(* IEC 61131-3 sources: volt/packages/volt-lsp-iec/test-corpus/bakon-nano/Device/Plc Logic/Application/POUs/FunctionBlocksAGM, 5 files *)

(* ---- ReadParametersFromAGM.pou ---- *)
FUNCTION_BLOCK ReadParametersFromAGM
VAR
	byStepper: BYTE;
	R_TRIG1: R_TRIG;
	bStartRead: BOOL;
	R_TRIG2: R_TRIG;
	LenzeParRead_LDC1: CIA405.SDO_READ4; (*TODO aanroep fixen CAA_Cia_405 en dan SDO_READ4*)
	Device : CIA405.DEVICE := 21;
	BLINK1: BLINK;
	TON1 :TON;
	byMasterNumber:BYTE:= 1;
	ptrByteArray : POINTER TO ARRAY[0..3] OF BYTE;
END_VAR
VAR_INPUT
	I_bEnable:BOOL;
END_VAR
VAR_OUTPUT
	bReady: BOOL;
END_VAR
VAR_IN_OUT
	Q_dwAGM_Status			: DWORD;
	Q_dwAGM_PowerLoss	: DWORD;
	Q_dwAGM_Frequency	: REAL;
	Q_dwAGM_ID				: DWORD;
END_VAR

%LANGUAGE ST
(*Create toggle for reading the parameters*)
BLINK1		(ENABLE:=I_bEnable ,
				 TIMELOW:=t#6s ,
				TIMEHIGH:=t#100ms,
				OUT=> );
R_TRIG1(CLK:=BLINK1.OUT);

IF R_TRIG1.Q THEN
	bStartRead:=TRUE;
END_IF

R_TRIG2(CLK:=LenzeParRead_LDC1.ERROR <> CIA405.CANOPEN_KERNEL_ERROR.CANOPEN_KERNEL_NO_ERROR);// OR LenzeParRead_LDC1.xTimeOut);(*TODO*)

IF NOT bStartRead OR R_TRIG2.Q OR NOT I_bEnable THEN
	byStepper:=0;
	bReady:=FALSE;
	bStartRead:=FALSE;
	LenzeParRead_LDC1(ENABLE:=FALSE);
	Q_dwAGM_ID := 0;
ELSE
	(*Alleen tijdens opstarten uitlezen*)
	CASE byStepper OF
	0:	(*Reset write FB*)
		bReady:=FALSE;
		TON1(IN:= FALSE);
		byStepper:=1;

	(*index 2003, generator status*)
	1:	LenzeParRead_LDC1(
		ENABLE:= FALSE,
		NETWORK :=byMasterNumber,
		Device:= Device,		 (* Adresse des Reglers *)
		Index:=8195,					(* Code *)
		SUBIndex:=0);				(* SubCode *)
		byStepper:=2;

	2:	LenzeParRead_LDC1(ENABLE:=TRUE,
								NETWORK:=ByMasterNumber);
		IF LenzeParRead_LDC1.CONFIRM THEN
			ptrByteArray := ADR(Q_dwAGM_Status);
			ptrByteArray^[0] := LenzeParRead_LDC1.DATA[1];
			ptrByteArray^[1] := LenzeParRead_LDC1.DATA[2];
			ptrByteArray^[2] := LenzeParRead_LDC1.DATA[3];
			ptrByteArray^[3] := LenzeParRead_LDC1.DATA[4];
			//Q_dwAGM_Status := SHL(SHL(SHL(LenzeParRead_LDC1.DATA[4],8) OR LenzeParRead_LDC1.DATA[3],8) OR LenzeParRead_LDC1.DATA[2],8) OR LenzeParRead_LDC1.DATA[1];	(* Codestelle wird gelesen *)
			LenzeParRead_LDC1(ENABLE:=FALSE);
			byStepper:=6;
		END_IF

	(*index 2008, Power loss*)
	6:	LenzeParRead_LDC1(
		ENABLE:= FALSE,
		Device:= Device,			(* Adresse des Reglers *)
		Index:=8200,						(* Code *)
		SubIndex:=0);					(* SubCode *)
		TON1(IN:=TRUE, PT:= t#1000ms);
		IF TON1.Q THEN
			byStepper:=8;
			TON1(IN:= FALSE);
		END_IF

	8:	LenzeParRead_LDC1(ENABLE:=TRUE,
								NETWORK:=1 );
		IF LenzeParRead_LDC1.CONFIRM THEN
			ptrByteArray := ADR(Q_dwAGM_PowerLoss);
			ptrByteArray^[0] := LenzeParRead_LDC1.DATA[1];
			ptrByteArray^[1] := LenzeParRead_LDC1.DATA[2];
			ptrByteArray^[2] := LenzeParRead_LDC1.DATA[3];
			ptrByteArray^[3] := LenzeParRead_LDC1.DATA[4];
			//Q_dwAGM_PowerLoss :=SHL(SHL(SHL(LenzeParRead_LDC1.DATA[4],8) OR LenzeParRead_LDC1.DATA[3],8) OR LenzeParRead_LDC1.DATA[2],8) OR LenzeParRead_LDC1.DATA[1];	(* Codestelle wird gelesen *)
			LenzeParRead_LDC1(ENABLE:=FALSE);
			byStepper:=12;
		END_IF

	(*index 2009, weld frequency*)
	12:	LenzeParRead_LDC1(
		Enable:= FALSE,
		NETWORK:=1,
		DEVICE:= Device,		(* Adresse des Reglers *)
		INDEX:=8201,					(* Code *)
		SUBINDEX:=0);				(* SubCode *)
		TON1(IN:=TRUE, PT:= t#1000ms);
		IF TON1.Q THEN
			byStepper:=14;
			TON1(IN:= FALSE);
		END_IF

	14:LenzeParRead_LDC1(ENABLE:=TRUE,
								NETWORK:=1);
		IF LenzeParRead_LDC1.CONFIRM THEN
			ptrByteArray := ADR(Q_dwAGM_Frequency);
			ptrByteArray^[0] := LenzeParRead_LDC1.DATA[1];
			ptrByteArray^[1] := LenzeParRead_LDC1.DATA[2];
			ptrByteArray^[2] := LenzeParRead_LDC1.DATA[3];
			ptrByteArray^[3] := LenzeParRead_LDC1.DATA[4];
			//Q_dwAGM_Frequency :=SHL(SHL(SHL(LenzeParRead_LDC1.DATA[4],8) OR LenzeParRead_LDC1.DATA[3],8) OR LenzeParRead_LDC1.DATA[2],8) OR LenzeParRead_LDC1.DATA[1];	(* Codestelle wird gelesen *)
			LenzeParRead_LDC1(ENABLE:=FALSE);
			byStepper:=20;
		END_IF

	(* Inlezen code 1018 (Vendor ID) Als deze 0 dan is er dus geen communicatie *)
	(*index 1018, Vendor ID *)
	20:	LenzeParRead_LDC1(
		Enable:= FALSE,
		NETWORK:=1,
		DEVICE:= Device,		(* Adresse des Reglers *)
		INDEX:=4120,						(* Code *)
		SUBINDEX:=1);					(* SubCode *)
		TON1(IN:=TRUE, PT:= t#1000ms);
		IF TON1.Q THEN
			byStepper:=22;
			TON1(IN:= FALSE);
		END_IF

	22:	LenzeParRead_LDC1(ENABLE:=TRUE,
								NETWORK:=1 );
		IF LenzeParRead_LDC1.CONFIRM THEN
			ptrByteArray := ADR(Q_dwAGM_ID);
			ptrByteArray^[0] := LenzeParRead_LDC1.DATA[1];
			ptrByteArray^[1] := LenzeParRead_LDC1.DATA[2];
			ptrByteArray^[2] := LenzeParRead_LDC1.DATA[3];
			ptrByteArray^[3] := LenzeParRead_LDC1.DATA[4];
			//Q_dwAGM_ID :=SHL(SHL(SHL(LenzeParRead_LDC1.DATA[4],8) OR LenzeParRead_LDC1.DATA[3],8) OR LenzeParRead_LDC1.DATA[2],8) OR LenzeParRead_LDC1.DATA[1];	(* Codestelle wird gelesen *)
			LenzeParRead_LDC1(ENABLE:=FALSE);
			byStepper:=30;
		END_IF

	30:	bReady:=TRUE;
		bStartRead:=FALSE;

	END_CASE

END_IF

END_FUNCTION_BLOCK

(* ---- StatusAGM.pou ---- *)
FUNCTION_BLOCK StatusAGM
VAR_INPUT
	I_dwAGM_Status: DWORD;
END_VAR
VAR_OUTPUT
	Q_dwErrorDetailsAGM	: DWORD;
	Q_bError					: BOOL;
END_VAR

%LANGUAGE ST
(*************************************************************************
 *
 * Application name			: Snijmachine met ultrasoon generator
 * Module name				: StatusAGM
 * Version number module	: 1.10
 *
 *
 *                  Copyright (c) Bakon 2009
 *                  Goes, The Netherlands
 *
 *
 * All rights are reserved. Reproduction in whole or in part is prohibited
 * without the written consent of the copyright owner.
 *
 *************************************************************************)

(*************************************************************************
 * HISTORY
 *************************************************************************
 * Update  :  1.1
 * Author  :    K. Kole
 * Changes : Q_bError bit added
 *************************************************************************)

(* Status ultrasoon generator *)
Q_bError	:= FALSE;
IF I_dwAGM_Status <> 0 THEN
	IF I_dwAGM_Status.0 THEN		(* SupplyVoltagetoLow *)
		Q_dwErrorDetailsAGM		:= 1;
		Q_bError	:= TRUE;
	ELSIF I_dwAGM_Status.1 THEN	(* Internal12VoltError *)
		Q_dwErrorDetailsAGM		:= 2;
		Q_bError	:= TRUE;
	ELSIF I_dwAGM_Status.2 THEN	(* Minimal PWM level reached *)
		Q_dwErrorDetailsAGM		:= 3;
		Q_bError	:= TRUE;
	ELSIF I_dwAGM_Status.3 THEN	(* Temperaure too high *)
		Q_dwErrorDetailsAGM		:= 4;
		Q_bError	:= TRUE;
	ELSIF I_dwAGM_Status.8 THEN	(* Frequency too low *)
		Q_dwErrorDetailsAGM		:= 5;
		Q_bError	:= TRUE;
	ELSIF I_dwAGM_Status.9 THEN	(* Frequency too high *)
		Q_dwErrorDetailsAGM		:= 6;
		Q_bError	:= TRUE;
	ELSIF I_dwAGM_Status.10 THEN	(* Maximum converter voltage reached *)
		Q_dwErrorDetailsAGM		:= 7;
		Q_bError	:= TRUE;
	ELSIF I_dwAGM_Status.11 THEN	(* Power overload *)
		Q_dwErrorDetailsAGM		:= 8;
		Q_bError	:= TRUE;
	ELSIF I_dwAGM_Status.12 THEN	(* Maximum PWM level reached *)
		Q_dwErrorDetailsAGM		:= 9;
		Q_bError	:= TRUE;
	ELSIF I_dwAGM_Status.13 THEN	(* No converter connected *)
		Q_dwErrorDetailsAGM		:= 10;
		Q_bError	:= TRUE;
	ELSIF I_dwAGM_Status.16 THEN	(* Minimum energy limit error *)
		Q_dwErrorDetailsAGM		:= 11;
		Q_bError	:= TRUE;
	ELSIF I_dwAGM_Status.17 THEN	(* Maximum energy limit error *)
		Q_dwErrorDetailsAGM		:= 12;
		Q_bError	:= TRUE;
	ELSIF I_dwAGM_Status.18 THEN	(* Minimum time limit error *)
		Q_dwErrorDetailsAGM		:= 13;
		Q_bError	:= TRUE;
	ELSIF I_dwAGM_Status.19 THEN	(* Maximum time limit error *)
		Q_dwErrorDetailsAGM		:= 14;
		Q_bError	:= TRUE;
	ELSIF I_dwAGM_Status.20 THEN	(* Minimum power limit error *)
		Q_dwErrorDetailsAGM		:= 15;
		Q_bError	:= TRUE;
	ELSIF I_dwAGM_Status.21 THEN	(* Maximum power limit error *)
		Q_dwErrorDetailsAGM		:= 16;
		Q_bError	:= TRUE;
	ELSIF I_dwAGM_Status.22 THEN	(* External analog amplitude too low *)
		Q_dwErrorDetailsAGM		:= 17;
		Q_bError	:= TRUE;
	ELSIF I_dwAGM_Status.30 THEN	(* Ultrasonic was stopped irregularly *)
		Q_dwErrorDetailsAGM		:= 18;
		Q_bError	:= TRUE;
	ELSIF I_dwAGM_Status.31 THEN	(* Ultrasonic active *)
		Q_dwErrorDetailsAGM		:= 19;
	ELSE
		Q_dwErrorDetailsAGM		:= 0;
	END_IF
ELSE
		Q_dwErrorDetailsAGM		:= 0;
END_IF

END_FUNCTION_BLOCK

(* ---- WriteControlRegAGM.pou ---- *)
FUNCTION_BLOCK WriteControlRegAGM
VAR
	byStepper: BYTE;
	bStartWrite: BOOL;
	R_TRIG1: R_TRIG;
	byControlRegAGM: BYTE;
	LenzeParWrite_LDC1: CIA405.SDO_WRITE4;
	dSendData : DWORD;
	DataArray : ARRAY[1..4] OF BYTE;
	ptrByteArray : POINTER TO ARRAY[0..3] OF BYTE;
END_VAR

VAR_INPUT
	byNodeID: BYTE;
	bStartAGM: BOOL;
	bStopAGM: BOOL;
	bTestAGM: BOOL;
END_VAR

%LANGUAGE ST
(*de index 2000 het control register wordt beschreven*)

R_TRIG1(CLK:=bStartAGM OR bStopAGM OR bTestAGM);

(*convert digital inputs to byte for control word*)
IF bStartAGM AND NOT bStopAGM AND NOT bTestAGM THEN
	byControlRegAGM:=1;
ELSIF NOT bStartAGM AND NOT bStopAGM AND bTestAGM THEN
	byControlRegAGM:=4;
ELSE			(*IF NOT bStartAGM AND bStopAGM AND NOT bTestAGM THEN*)
	byControlRegAGM:=2;
END_IF

IF R_TRIG1.Q THEN
	bStartWrite:=TRUE;
END_IF

IF NOT bStartWrite  THEN
	byStepper:=0;
ELSE

	CASE byStepper OF
	0:	(*Reset write FB*)
		LenzeParWrite_LDC1(ENABLE:=FALSE);
		byStepper:=1;

	(*index 2000 control register*)
	1:	dSendData := BYTE_TO_DWORD(byControlRegAGM);
		ptrByteArray := ADR(dSendData);
		DataArray[1] := ptrByteArray^[0];
		DataArray[2] := ptrByteArray^[1];
		DataArray[3] := ptrByteArray^[2];
		DataArray[4] := ptrByteArray^[3];
		LenzeParWrite_LDC1(
		ENABLE:=FALSE ,
		DEVICE:=byNodeID ,					(* Adresse des Reglers *)
		NETWORK:=1,
		INDEX:=8192 ,
		SUBINDEX:=0 ,					(* SubCode *)

		DATA:= DataArray,//BYTE_TO_DWORD(byControlRegAGM),
		DataLength:=1);
		byStepper:=2;

	2:	LenzeParWrite_LDC1(ENABLE:=TRUE, NETWORK:=1);
		IF LenzeParWrite_LDC1.CONFIRM OR (LenzeParWrite_LDC1.ERROR <> CIA405.CANOPEN_KERNEL_ERROR.CANOPEN_KERNEL_NO_ERROR)THEN
			LenzeParWrite_LDC1(ENABLE:=FALSE);
			bStartWrite:=FALSE;
			byStepper:=0;
		END_IF

	END_CASE

END_IF

END_FUNCTION_BLOCK

(* ---- WriteParametersToAGM.pou ---- *)
FUNCTION_BLOCK WriteParametersToAGM
VAR
	byStepper: BYTE;
	bStartWrite: BOOL;
	R_TRIG1: R_TRIG;
	R_TRIG2: R_TRIG;
	LenzeParWrite_LDC1: CIA405.SDO_WRITE4; (*TODO -> Hoe Axis ref hiervoor maken?*)
	Device : CIA405.DEVICE := 21;
	DataArray : ARRAY[1..4] OF BYTE;
	ptrByteArray : POINTER TO ARRAY[0..3] OF BYTE;
END_VAR
VAR_INPUT
	I_bEnable		: BOOL;
	I_dwAGM_Amplitude	: DWORD;
END_VAR

%LANGUAGE ST
(*de index 2000 control register en index 2010 de amplitude worden beschreven*)

R_TRIG1(CLK:=I_bEnable);

IF R_TRIG1.Q THEN
	bStartWrite:=TRUE;
END_IF

R_TRIG2(CLK:=LenzeParWrite_LDC1.ERROR <> CIA405.CANOPEN_KERNEL_ERROR.CANOPEN_KERNEL_NO_ERROR);

IF NOT bStartWrite OR R_TRIG2.Q THEN
	bStartWrite:=FALSE;
	byStepper:=0;
	//LenzeParWrite_LDC1(ENABLE := FALSE);
ELSE

	CASE byStepper OF
	0:	(*Reset write FB*)
		LenzeParWrite_LDC1(ENABLE:=FALSE);
		byStepper:=1;

	(*index 2010 weld amplitude*)
	1:	ptrByteArray := ADR(I_dwAGM_Amplitude);
		DataArray[4] := ptrByteArray^[3];
		DataArray[3] := ptrByteArray^[2];
		DataArray[2] := ptrByteArray^[1];
		DataArray[1] := ptrByteArray^[0];
		LenzeParWrite_LDC1(
		ENABLE	:=FALSE ,
		DEVICE	:= Device,			(* Adresse des Reglers *)
		NETWORK:=1,
		INDEX		:=8208 ,
		SUBINDEX:=0 ,					(* SubCode *)
		DATA:=DataArray,
		DATALENGTH:=1 );
		byStepper:=2;

	2:	LenzeParWrite_LDC1(ENABLE:=TRUE,
		NETWORK:=1);
		IF LenzeParWrite_LDC1.CONFIRM THEN
			bStartWrite:=FALSE;
			byStepper:=0;
		END_IF
	END_CASE

END_IF

END_FUNCTION_BLOCK

(* ---- CanBridgeAGM.pou ---- *)
PROGRAM CanBridgeAGM
VAR
END_VAR

%LANGUAGE ST
//Set bus variables to local
g_dwAGM1_PowerLoss 							:= CAN_TO_PLC.dwAGM1_PowerLoss;
g_rAGM1_Frequency 							:= CAN_TO_PLC.rAGM1_Frequency;
g_sMACH.ERR.bAGM1_CommFailure 				:= CAN_TO_PLC.bAGM1_CommFailure;
g_sHMI_Mach_UnitStatus.dwErrorDetailsAGM1 	:= CAN_TO_PLC.dwErrorDetailsAGM1;
g_sMACH.ERR.bUltrasonic1					 := CAN_TO_PLC.bUltrasonic1;

//Set local variables to the bus
PLC_TO_CAN.g_bOnDelayed 								:= g_bOnDelayed;
PLC_TO_CAN.g_bDQ_Ultrasonic1 							:= g_bDQ_Ultrasonic1;
PLC_TO_CAN.g_bTestAGM1									:= g_bTestAGM1;
PLC_TO_CAN.g_HMI_MachCommand.bScanMode					:= g_HMI_MachCommand.bScanMode;
PLC_TO_CAN.g_HMI_RCP_Parameters.dwUltrasonicPower1		:= g_HMI_RCP_Parameters.dwUltrasonicPower1;
PLC_TO_CAN.g_HMI_MCH_Parameters.bUltrasonicEnable1		:= g_HMI_MCH_Parameters.bUltrasonicEnable1;
PLC_TO_CAN.C_rMaxPowerUS1								:= C_rMaxPowerUS1;

END_PROGRAM
